FUNCTION_BLOCK Arm
  (* Version 0.1, 2005-04-08, Author Name, Chalmers *)
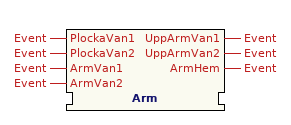
  EVENT_INPUT
    PlockaVan1;
    PlockaVan2;
    ArmVan1;
    ArmVan2;
  END_EVENT
  EVENT_OUTPUT
    UppArmVan1;
    UppArmVan2;
    ArmHem;
  END_EVENT
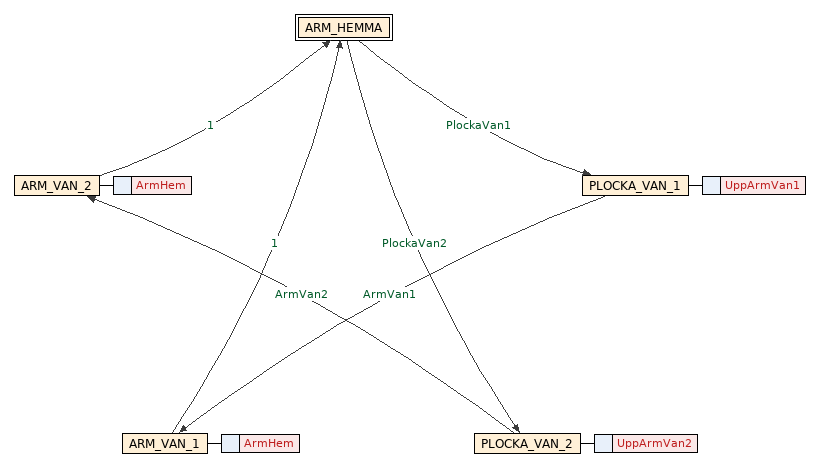
  EC_STATES
    ARM_HEMMA;
    PLOCKA_VAN_1 : -> UppArmVan1;
    PLOCKA_VAN_2 : -> UppArmVan2;
    ARM_VAN_1 : -> ArmHem;
    ARM_VAN_2 : -> ArmHem;
  END_STATES
  EC_TRANSITIONS
    ARM_HEMMA TO PLOCKA_VAN_1 := PlockaVan1;
    ARM_HEMMA TO PLOCKA_VAN_2 := PlockaVan2;
    PLOCKA_VAN_1 TO ARM_VAN_1 := ArmVan1;
    PLOCKA_VAN_2 TO ARM_VAN_2 := ArmVan2;
    ARM_VAN_1 TO ARM_HEMMA := 1;
    ARM_VAN_2 TO ARM_HEMMA := 1;
  END_TRANSITIONS
END_FUNCTION_BLOCK
